{attribute 'GeneratedUsingTerminal: EP7041-0002-0018'}
{attribute addProperty BoxType "EP7041-0002-0018"}
{attribute addProperty Id "AdsAddrAT %I*.TcoAmsAddr0Chn0AT %I*USINT1Chn1AT %I*USINT1StateAT %I*UINT2"}
{attribute addProperty CRC "995053194"}
{attribute addProperty Size "4"}
TYPE InfoData_3B4F4E8A EXTENDS InputBase_8311D824 :
STRUCT
	{attribute addProperty Name "AdsAddr"}
	AdsAddr AT %I* : .TcoAmsAddr;
	{attribute addProperty Name "Chn0"}
	Chn0 AT %I* : USINT;
	{attribute addProperty Name "Chn1"}
	Chn1 AT %I* : USINT;
	{attribute addProperty Name "State"}
	State AT %I* : UINT;
END_STRUCT
END_TYPE

(* stored: Version 1.2.0.0, ProductVersion 3.1.4024.9
   DUT InfoData_3B4F4E8A: Id {c130683e-fd5a-4e0f-9e22-dd644cd9d081} *)
